PROGRAM MAIN
VAR
END_VAR

END_PROGRAM

(* stored: Version 1.1.0.1
   POU MAIN: Id {0b4cac4f-6a1c-4ecc-b962-dc24e9c4fc60} *)
